{attribute 'GeneratedUsingTerminal: CU1124-0000-0016'}
{attribute addProperty BoxType "CU1124-0000-0016"}
{attribute addProperty Id "A_0004_CU1128_0000_0000A_0004_CU1128_0000_0000_2F60DA9F124"}
{attribute addProperty CRC "3463119944"}
{attribute addProperty Size "124"}
TYPE A_0003_CU1124_0000_0016_CE6B0448 EXTENDS CU1124_1FC0878B :
STRUCT
	{attribute addProperty Name "A_0004(CU1128-0000-0000)"}
	{attribute addProperty PreviousPort "A_0003(CU1124-0000-0016) : D"}
	A_0004_CU1128_0000_0000 : A_0004_CU1128_0000_0000_2F60DA9F;
END_STRUCT
END_TYPE

(* stored: Version 1.2.0.0, ProductVersion 3.1.4024.9
   DUT A_0003_CU1124_0000_0016_CE6B0448: Id {d0a0f981-e195-4472-99ce-92aacde21a2c} *)
